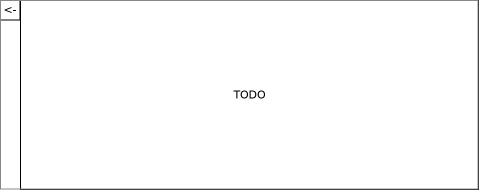
VISUALIZATION _VISU_MarkCamera  // 479x190
    RoundedRectangle (0,0 20x20), "<-"
        OnMouseClick: change screen: Previous 
    Rectangle (20,0 459x190), "TODO"
END_VISUALIZATION

(* stored: Version 1.1.0.1, ProductVersion 3.1.4024.3
   Visu _VISU_MarkCamera: Id {fad9d89a-4ff7-4110-8451-a36de41742f7} *)
